KUKA KRL program: flexion2.src, flexion2.dat

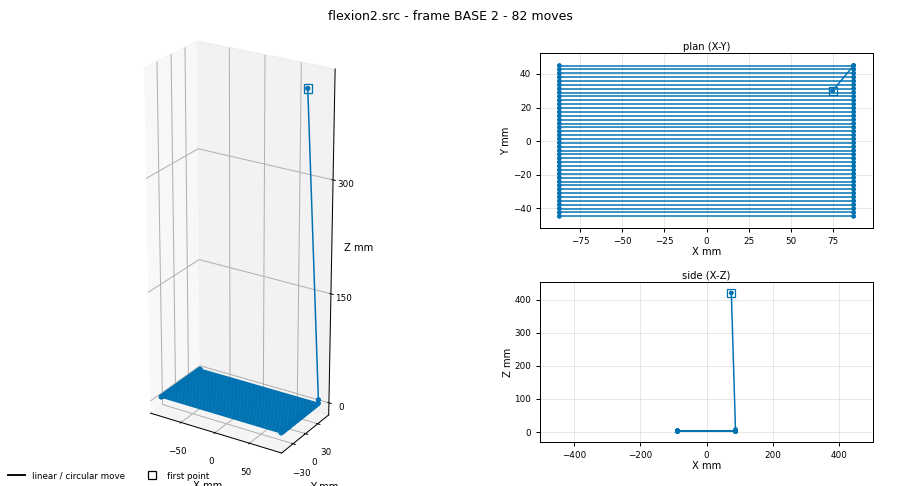
[picture p0: tool path of flexion2.src in frame BASE 2, 82 of 84 moves have a stored position in this frame; points joined in program order, loops and branches not executed]
--- flexion2.src ---
&ACCESS RVP
&PARAM TEMPLATE = C:\KRC\Roboter\Template\vorgabe
&PARAM EDITMASK = *
DEF flexion2( )
;FOLD INI;%{PE}%V3.2.0,%MKUKATPBASIS,%CINIT,%VCOMMON,%P
;FOLD BAS INI;%{E}%V3.2.0,%MKUKATPBASIS,%CINIT,%VINIT,%P
GLOBAL INTERRUPT DECL 3 WHEN $STOPMESS==TRUE DO IR_STOPM ( )
INTERRUPT ON 3
BAS (#INITMOV,0 )
;ENDFOLD (BAS INI)
;FOLD A20 INI;%{E}%V3.2.0,%MKUKATPA20,%CINIT,%VINIT,%P
IF ARC20==TRUE THEN
A20 (ARC_INI)
INTERRUPT DECL 6 WHEN $CYCFLAG[3]==FALSE DO A20(TECH_STOP2)
ENDIF
;ENDFOLD (A20 INI)
;FOLD A10 INI;%{E}%V3.2.0,%MKUKATPARC,%CINIT,%VINIT,%P
IF A10_OPTION==#ACTIVE THEN
INTERRUPT DECL 4 WHEN $CYCFLAG[2]==FALSE DO A10 (#APPL_ERROR)
INTERRUPT DECL 7 WHEN A_ARC_SWI==#ACTIVE DO A10 (#ARC_SEAM)
INTERRUPT DECL 5 WHEN A_FLY_ARC==TRUE DO A10 (#HPU_ARC)
INTERRUPT  ON 5
A10_INI ( )
ENDIF
;ENDFOLD (A10 INI)
;FOLD GRIPPER INI;%{E}%V3.2.0,%MKUKATPGRIPPER,%CINIT,%VINIT,%P
USER_GRP(0,DUMMY,DUMMY,GDEFAULT)
;ENDFOLD (GRIPPER INI)
;FOLD SPOT INI;%{E}%V3.2.0,%MKUKATPSPOT,%CINIT,%VINIT,%P
USERSPOT(#INIT)
;ENDFOLD (SPOT INI)
;FOLD TOUCHSENSE INI;%{E}%V3.2.0,%MKUKATPTS,%CINIT,%VINIT,%P
IF H70_OPTION THEN
INTERRUPT DECL 15 WHEN $MEAS_PULSE[TOUCH_I[TOUCH_ACTIVE].IN_NR] DO H70 (6,CD0 )
INTERRUPT DECL 16 WHEN $ZERO_MOVE DO H70 (7,CD0 )
INTERRUPT DECL 17 WHEN $TECHPAR_C[FG_TOUCH,8]>0.5 DO H70 (8,CD0)
H70 (1,CD0 )
ENDIF
;ENDFOLD (TOUCHSENSE INI)
;FOLD USER INI;%{E}%V3.2.0,%MKUKATPUSER,%CINIT,%VINIT,%P
;Make your modifications here
;ENDFOLD (USER INI)
;ENDFOLD (INI)
; SPEED PTP FOR AXIS
$VEL_AXIS[1] = 15
$VEL_AXIS[2] = 15
$VEL_AXIS[3] = 15
$VEL_AXIS[4] = 15
$VEL_AXIS[5] = 15
$VEL_AXIS[6] = 15
;SMOOTHNESS
$APO.CDIS = 2
;ADVANCE
$ADVANCE = 3
;SET TOOL AND BASE
$TOOL = TOOL_DATA[3]
$BASE = BASE_DATA[2]
;HOME
;FOLD PTP HOME Vel=10% DEFAULT
$BWDSTART=FALSE
$H_POS=XHOME
PDAT_ACT=PDEFAULT
FDAT_ACT=FHOME
BAS(#PTP_DAT )
BAS (#VEL_PTP,10 )
PTP XHOME
;ENDFOLD
;USER PROGRAM
;SPEED $VEL.CP
$VEL.CP=0.03
; OUT[TEMP] = 200
; OUT[vent] = 1
; OUT[RPM] = 30
; USER POSES CALLS
PTP {X 75, Y 30, Z 420, A 0, B 90, C 0}
; USER POSES CALLS
LIN {X 87.5, Y 45.0, Z 7.5, A 0, B 90, C 0} C_DIS
WAIT SEC 1
$OUT[1] = TRUE
LIN {X 87.5, Y 45.0, Z 2.5, A 0, B 90, C 0} C_DIS
LIN {X -87.5, Y 45.0, Z 2.5, A 0, B 90, C 0} C_DIS
LIN {X -87.5, Y 42.7, Z 2.5, A 0, B 90, C 0} C_DIS
LIN {X 87.5, Y 42.7, Z 2.5, A 0, B 90, C 0} C_DIS
LIN {X 87.5, Y 40.4, Z 2.5, A 0, B 90, C 0} C_DIS
LIN {X -87.5, Y 40.4, Z 2.5, A 0, B 90, C 0} C_DIS
LIN {X -87.5, Y 38.1, Z 2.5, A 0, B 90, C 0} C_DIS
LIN {X 87.5, Y 38.1, Z 2.5, A 0, B 90, C 0} C_DIS
LIN {X 87.5, Y 35.8, Z 2.5, A 0, B 90, C 0} C_DIS
LIN {X -87.5, Y 35.8, Z 2.5, A 0, B 90, C 0} C_DIS
LIN {X -87.5, Y 33.5, Z 2.5, A 0, B 90, C 0} C_DIS
LIN {X 87.5, Y 33.5, Z 2.5, A 0, B 90, C 0} C_DIS
LIN {X 87.5, Y 31.2, Z 2.5, A 0, B 90, C 0} C_DIS
LIN {X -87.5, Y 31.2, Z 2.5, A 0, B 90, C 0} C_DIS
LIN {X -87.5, Y 28.9, Z 2.5, A 0, B 90, C 0} C_DIS
LIN {X 87.5, Y 28.9, Z 2.5, A 0, B 90, C 0} C_DIS
LIN {X 87.5, Y 26.6, Z 2.5, A 0, B 90, C 0} C_DIS
LIN {X -87.5, Y 26.6, Z 2.5, A 0, B 90, C 0} C_DIS
LIN {X -87.5, Y 24.3, Z 2.5, A 0, B 90, C 0} C_DIS
LIN {X 87.5, Y 24.3, Z 2.5, A 0, B 90, C 0} C_DIS
LIN {X 87.5, Y 22.0, Z 2.5, A 0, B 90, C 0} C_DIS
LIN {X -87.5, Y 22.0, Z 2.5, A 0, B 90, C 0} C_DIS
LIN {X -87.5, Y 19.7, Z 2.5, A 0, B 90, C 0} C_DIS
LIN {X 87.5, Y 19.7, Z 2.5, A 0, B 90, C 0} C_DIS
LIN {X 87.5, Y 17.4, Z 2.5, A 0, B 90, C 0} C_DIS
LIN {X -87.5, Y 17.4, Z 2.5, A 0, B 90, C 0} C_DIS
LIN {X -87.5, Y 15.1, Z 2.5, A 0, B 90, C 0} C_DIS
LIN {X 87.5, Y 15.1, Z 2.5, A 0, B 90, C 0} C_DIS
LIN {X 87.5, Y 12.8, Z 2.5, A 0, B 90, C 0} C_DIS
LIN {X -87.5, Y 12.8, Z 2.5, A 0, B 90, C 0} C_DIS
LIN {X -87.5, Y 10.5, Z 2.5, A 0, B 90, C 0} C_DIS
LIN {X 87.5, Y 10.5, Z 2.5, A 0, B 90, C 0} C_DIS
LIN {X 87.5, Y 8.2, Z 2.5, A 0, B 90, C 0} C_DIS
LIN {X -87.5, Y 8.2, Z 2.5, A 0, B 90, C 0} C_DIS
LIN {X -87.5, Y 5.9, Z 2.5, A 0, B 90, C 0} C_DIS
LIN {X 87.5, Y 5.9, Z 2.5, A 0, B 90, C 0} C_DIS
LIN {X 87.5, Y 3.6, Z 2.5, A 0, B 90, C 0} C_DIS
LIN {X -87.5, Y 3.6, Z 2.5, A 0, B 90, C 0} C_DIS
LIN {X -87.5, Y 1.3, Z 2.5, A 0, B 90, C 0} C_DIS
LIN {X 87.5, Y 1.3, Z 2.5, A 0, B 90, C 0} C_DIS
LIN {X 87.5, Y -1.0, Z 2.5, A 0, B 90, C 0} C_DIS
LIN {X -87.5, Y -1.0, Z 2.5, A 0, B 90, C 0} C_DIS
LIN {X -87.5, Y -3.3, Z 2.5, A 0, B 90, C 0} C_DIS
LIN {X 87.5, Y -3.3, Z 2.5, A 0, B 90, C 0} C_DIS
LIN {X 87.5, Y -5.6, Z 2.5, A 0, B 90, C 0} C_DIS
LIN {X -87.5, Y -5.6, Z 2.5, A 0, B 90, C 0} C_DIS
LIN {X -87.5, Y -7.9, Z 2.5, A 0, B 90, C 0} C_DIS
LIN {X 87.5, Y -7.9, Z 2.5, A 0, B 90, C 0} C_DIS
LIN {X 87.5, Y -10.2, Z 2.5, A 0, B 90, C 0} C_DIS
LIN {X -87.5, Y -10.2, Z 2.5, A 0, B 90, C 0} C_DIS
LIN {X -87.5, Y -12.5, Z 2.5, A 0, B 90, C 0} C_DIS
LIN {X 87.5, Y -12.5, Z 2.5, A 0, B 90, C 0} C_DIS
LIN {X 87.5, Y -14.8, Z 2.5, A 0, B 90, C 0} C_DIS
LIN {X -87.5, Y -14.8, Z 2.5, A 0, B 90, C 0} C_DIS
LIN {X -87.5, Y -17.1, Z 2.5, A 0, B 90, C 0} C_DIS
LIN {X 87.5, Y -17.1, Z 2.5, A 0, B 90, C 0} C_DIS
LIN {X 87.5, Y -19.4, Z 2.5, A 0, B 90, C 0} C_DIS
LIN {X -87.5, Y -19.4, Z 2.5, A 0, B 90, C 0} C_DIS
LIN {X -87.5, Y -21.7, Z 2.5, A 0, B 90, C 0} C_DIS
LIN {X 87.5, Y -21.7, Z 2.5, A 0, B 90, C 0} C_DIS
LIN {X 87.5, Y -24.0, Z 2.5, A 0, B 90, C 0} C_DIS
LIN {X -87.5, Y -24.0, Z 2.5, A 0, B 90, C 0} C_DIS
LIN {X -87.5, Y -26.3, Z 2.5, A 0, B 90, C 0} C_DIS
LIN {X 87.5, Y -26.3, Z 2.5, A 0, B 90, C 0} C_DIS
LIN {X 87.5, Y -28.6, Z 2.5, A 0, B 90, C 0} C_DIS
LIN {X -87.5, Y -28.6, Z 2.5, A 0, B 90, C 0} C_DIS
LIN {X -87.5, Y -30.9, Z 2.5, A 0, B 90, C 0} C_DIS
LIN {X 87.5, Y -30.9, Z 2.5, A 0, B 90, C 0} C_DIS
LIN {X 87.5, Y -33.2, Z 2.5, A 0, B 90, C 0} C_DIS
LIN {X -87.5, Y -33.2, Z 2.5, A 0, B 90, C 0} C_DIS
LIN {X -87.5, Y -35.5, Z 2.5, A 0, B 90, C 0} C_DIS
LIN {X 87.5, Y -35.5, Z 2.5, A 0, B 90, C 0} C_DIS
LIN {X 87.5, Y -37.8, Z 2.5, A 0, B 90, C 0} C_DIS
LIN {X -87.5, Y -37.8, Z 2.5, A 0, B 90, C 0} C_DIS
LIN {X -87.5, Y -40.1, Z 2.5, A 0, B 90, C 0} C_DIS
LIN {X 87.5, Y -40.1, Z 2.5, A 0, B 90, C 0} C_DIS
LIN {X 87.5, Y -42.4, Z 2.5, A 0, B 90, C 0} C_DIS
LIN {X -87.5, Y -42.4, Z 2.5, A 0, B 90, C 0} C_DIS
LIN {X -87.5, Y -44.7, Z 2.5, A 0, B 90, C 0} C_DIS
LIN {X 87.5, Y -44.7, Z 2.5, A 0, B 90, C 0} C_DIS
$OUT[1] = FALSE

;Wait for
; END POSITION FOR
;END USER CODE
;HOME
;FOLD PTP HOME Vel=10% DEFAULT
$BWDSTART=FALSE
$H_POS=XHOME
PDAT_ACT=PDEFAULT
FDAT_ACT=FHOME
BAS(#PTP_DAT )
BAS (#VEL_PTP,10 )
PTP XHOME
;ENDFOLD
END

--- flexion2.dat ---
DEFDAT flexion2()
ENDDAT
